(* IEC 61131-3 sources: eCockpitGit/test_project/src/%F%00 Library/%F%Common Functions/%F%Y AXB/%F%Output, 6 files *)

(* ---- %POU%FU_lrABXToY.st ---- *)
//This function, calculates the y value in a y = a * x + b equation
// +-----------+----------+----------+-----------------------------------------------------------------------------------------------------------------------+
// |**Version**|**Author**| **Date** |**Changes**                                                                                                            |
// +-----------+----------+----------+-----------------------------------------------------------------------------------------------------------------------+
// | 1         | NSN      | 29-01-19 | Creation                                                                                                              |
// +-----------+----------+----------+-----------------------------------------------------------------------------------------------------------------------+
FUNCTION FU_lrABXToY : LREAL
VAR_INPUT
	rX		:LREAL;
	rA		:LREAL;
	rB		:LREAL;
END_VAR

(*%!%__DELIMITER__%!%*)
FU_lrABXToY	:=		rA * rX + rB;

(* ---- %POU%FU_lrABYToX.st ---- *)
//This function, calculates the x value in a x = (y - b) / a equation
// +-----------+----------+----------+-----------------------------------------------------------------------------------------------------------------------+
// |**Version**|**Author**| **Date** |**Changes**                                                                                                            |
// +-----------+----------+----------+-----------------------------------------------------------------------------------------------------------------------+
// | 1         | NSN      | 29-01-19 | Creation                                                                                                              |
// +-----------+----------+----------+-----------------------------------------------------------------------------------------------------------------------+
FUNCTION FU_lrABYToX : LREAL
VAR_INPUT
	rY		:LREAL;
	rA		:LREAL;
	rB		:LREAL;
END_VAR

(*%!%__DELIMITER__%!%*)
IF rA <> 0 THEN
	FU_lrABYToX	:=		(rY - rB) / rA;
ELSE
	FU_lrABYToX	:=		0;
END_IF

(* ---- %POU%FU_rABXToY.st ---- *)
//This function, calculates the y value in a y = a * x + b equation
// +-----------+----------+----------+-----------------------------------------------------------------------------------------------------------------------+
// |**Version**|**Author**| **Date** |**Changes**                                                                                                            |
// +-----------+----------+----------+-----------------------------------------------------------------------------------------------------------------------+
// | 1         | NSN      | 29-01-19 | Creation                                                                                                              |
// +-----------+----------+----------+-----------------------------------------------------------------------------------------------------------------------+
FUNCTION FU_rABXToY : REAL
VAR_INPUT
	rX		:REAL;
	rA		:REAL;
	rB		:REAL;
END_VAR

(*%!%__DELIMITER__%!%*)
FU_rABXToY	:=		rA * rX + rB;

(* ---- %POU%FU_rABXToYDP.st ---- *)
//This function, calculates the y value in a y = a * x + b equation
//This is the double precision version, which means all values are converted to LREAL before mathematics
// +-----------+----------+----------+-----------------------------------------------------------------------------------------------------------------------+
// |**Version**|**Author**| **Date** |**Changes**                                                                                                            |
// +-----------+----------+----------+-----------------------------------------------------------------------------------------------------------------------+
// | 1         | NSN      | 29-01-19 | Creation                                                                                                              |
// +-----------+----------+----------+-----------------------------------------------------------------------------------------------------------------------+
FUNCTION FU_rABXToYDP : REAL
VAR_INPUT
	rX		:REAL;
	rA		:REAL;
	rB		:REAL;
END_VAR

(*%!%__DELIMITER__%!%*)
FU_rABXToYDP	:=		TO_REAL(TO_LREAL(rA) * TO_LREAL(rX) + TO_LREAL(rB));

(* ---- %POU%FU_rABYToX.st ---- *)
//This function, calculates the x value in a x = (y - b) / a equation
// +-----------+----------+----------+-----------------------------------------------------------------------------------------------------------------------+
// |**Version**|**Author**| **Date** |**Changes**                                                                                                            |
// +-----------+----------+----------+-----------------------------------------------------------------------------------------------------------------------+
// | 1         | NSN      | 29-01-19 | Creation                                                                                                              |
// +-----------+----------+----------+-----------------------------------------------------------------------------------------------------------------------+
FUNCTION FU_rABYToX : REAL
VAR_INPUT
	rY		:REAL;
	rA		:REAL;
	rB		:REAL;
END_VAR

(*%!%__DELIMITER__%!%*)
IF rA <> 0 THEN
	FU_rABYToX	:=		(rY - rB) / rA;
ELSE
	FU_rABYToX	:=		0;
END_IF

(* ---- %POU%FU_rABYToXDP.st ---- *)
//This function, calculates the x value in a x = (y - b) / a equation
//This is the double precision version, which means all values are converted to LREAL before mathematics
// +-----------+----------+----------+-----------------------------------------------------------------------------------------------------------------------+
// |**Version**|**Author**| **Date** |**Changes**                                                                                                            |
// +-----------+----------+----------+-----------------------------------------------------------------------------------------------------------------------+
// | 1         | NSN      | 29-01-19 | Creation                                                                                                              |
// +-----------+----------+----------+-----------------------------------------------------------------------------------------------------------------------+
FUNCTION FU_rABYToXDP : REAL
VAR_INPUT
	rY		:REAL;
	rA		:REAL;
	rB		:REAL;
END_VAR

(*%!%__DELIMITER__%!%*)
IF rA <> 0 THEN
	FU_rABYToXDP	:=		TO_REAL((TO_LREAL(rY) - TO_LREAL(rB)) / TO_LREAL(rA));
ELSE
	FU_rABYToXDP	:=		0;
END_IF
